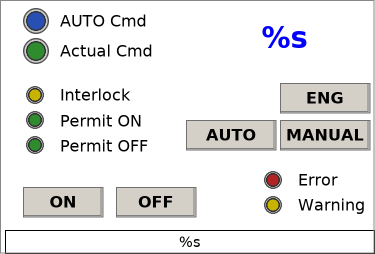
VISUALIZATION GUI_TEMPLATE_CMD_OVERRIDE  // 375x254
VAR_IN_OUT
	m_Cmd:		FB_CRYO_CMD_OVERRIDE;
END_VAR
    Lamp1 (25,85 20x20), variable: m_Cmd.out_bInterlock, style: Lamp-Lamp1-Yellow
    Lamp1 (25,110 20x20), variable: m_Cmd.bPermitOn, style: Lamp-Lamp1-Green
    Lamp1 (25,135 20x20), variable: m_Cmd.bPermitOff, style: Lamp-Lamp1-Green
    Rectangle (57,80 110x30), "Interlock"
    Rectangle (57,106 110x30), "Permit ON"
    Rectangle (57,131 110x30), "Permit OFF"
    Button (23,187 80x30), "ON", colour toggle: (m_Cmd.bPermitOn AND NOT m_Cmd.bAutoMode) OR m_Cmd.bEngMode, input disabled if: m_Cmd.bDisableBtnOn
        OnMouseClick: execute { m_Cmd.bManualCmd := TRUE; }
    Lamp1 (21,36 30x30), tooltip "Actual command going out", variable: m_Cmd.out_bEnable, style: Lamp-Lamp1-Green
    Rectangle (57,36 110x30), "Actual Cmd"
    Button (186,120 90x30), "AUTO", tooltip "Switch to AUTO Mode", colour toggle: m_Cmd.bAutoMode, input disabled if: m_Cmd.bAutoMode OR m_Cmd.bEngMode
        OnMouseClick: execute { m_Cmd.bAutoMode := TRUE; }
    Button (280,120 90x30), "MANUAL", tooltip "Switch to MANUAL Mode", colour toggle: NOT m_Cmd.bAutoMode, input disabled if: NOT m_Cmd.bAutoMode AND NOT m_Cmd.bEngMode
        OnMouseClick: execute { m_Cmd.bAutoMode := FALSE; }
    Button (116,187 80x30), "OFF", colour toggle: (m_Cmd.bPermitOff AND NOT m_Cmd.bAutoMode) OR m_Cmd.bEngMode, input disabled if: m_Cmd.bDisableBtnOff
        OnMouseClick: execute { m_Cmd.bManualCmd := FALSE; }
    Button (280,83 90x30), "ENG", tooltip "Toggle Engineering Mode", colour toggle: m_Cmd.bEngMode, input disabled if: m_Cmd.bAutoMode
        toggle m_Cmd.bEngMode
    Lamp1 (21,6 30x30), tooltip "Command coming from the Control System", variable: m_Cmd.in_bEnable, style: Lamp-Lamp1-Blue
    Rectangle (57,6 110x30), "AUTO Cmd"
    Rectangle (5,230 370x24), "%s", text variable: m_Cmd.out_sStatus
    Lamp1 (263,170 20x20), tooltip "If ON, there is an error in the SW implementation of permission handling.", variable: m_Cmd.out_bError, style: Lamp-Lamp1-Red
    Rectangle (295,165 75x30), "Error"
    Lamp1 (263,195 20x20), tooltip "If ON, ENG command is not safe!", variable: m_Cmd.out_bWarning, style: Lamp-Lamp1-Yellow
    Rectangle (295,190 75x30), "Warning"
    Rectangle (210,17 150x41), "%s", text variable: m_Cmd.out_sMode
END_VISUALIZATION

(* stored: Version 1.1.0.1, ProductVersion 3.1.4024.12
   Visu GUI_TEMPLATE_CMD_OVERRIDE: Id {bddcb5f1-918f-42a1-90a8-20d6676b2297} *)
